FUNCTION_BLOCK FB_ArrayExample

VAR
	test1 : ARRAY[GVL.INDEX_MIN..5] OF INT := [5,8, 9, 6, 7];
	test2 : ARRAY[1..10] OF INT := [10(8)]; // Will all be initalised with 8
	answer1, answer2 : DINT;
END_VAR

answer1 := M_SumArray(test1);
answer2 := M_SumArray(test2);

METHOD M_SumArray : DINT

VAR_IN_OUT
	data : ARRAY[*] OF INT;
END_VAR

VAR
	i, sum : DINT;
END_VAR
RETURN ( LEN2(DATA) < 1 );

FOR i := LOWER_BOUND(data, 1) TO UPPER_BOUND(data, 1) DO
	sum := sum + data[i];
END_FOR

M_SumArray := sum;
END_METHOD

END_FUNCTION_BLOCK

(* stored: Version 1.1.0.1
   POU FB_ArrayExample: Id {7cf751cb-8f08-4e56-9cfb-04114186b805}, SpecialFunc None
   Method M_SumArray: Id {11ca7274-3aea-480b-9ca4-580c591829db} *)
